KUKA KRL program: DisableRSI_Pos.src, DisableRSI_Pos.dat

--- DisableRSI_Pos.src ---
&ACCESS RV
&REL 1
DEF DisableRSI_Pos ( )
   $SEN_PINT[RSI_X_Sys_Disable]=1
END

--- DisableRSI_Pos.dat ---
&ACCESS RV
&REL 1
DEFDAT  DisableRSI_Pos PUBLIC

ENDDAT
